FUNCTION TryConvert_BOOL_TO_UINT : BOOL
VAR_INPUT
	in : BOOL;
	out : REFERENCE TO UINT;
END_VAR

out := BOOL_TO_UINT(in);
TryConvert_BOOL_TO_UINT := TRUE;

END_FUNCTION

(* stored: Version 1.1.0.1, ProductVersion 3.1.4024.12
   POU TryConvert_BOOL_TO_UINT: Id {e5cdf9a0-b81b-4fc2-a5e0-b0f42c3f6e26}, SpecialFunc None *)
